// TIA Portal V18 export
FUNCTION "HC_PIDs" : Void   // FC1019, LAD
{ S7_Optimized_Access := 'TRUE' }
VERSION : 0.1
// stored: AutoNumber false, IsIECCheckEnabled false, SetENOAutomatically false, UDAEnableTagReadback false
BEGIN

REGION Network 1
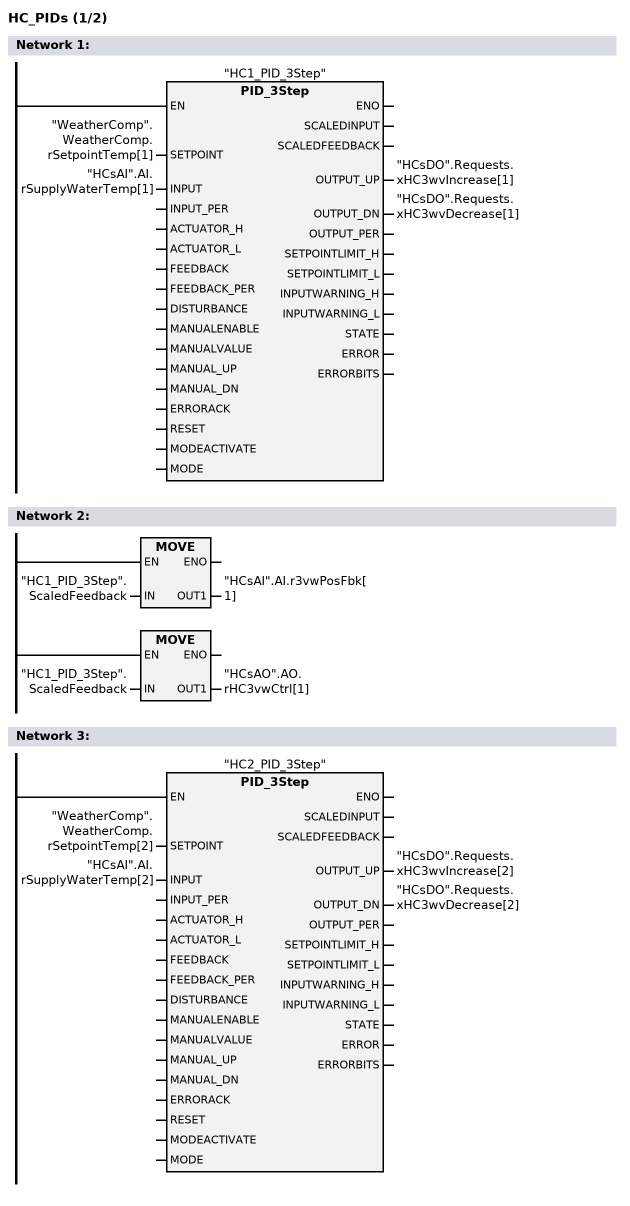
   RUNG wire#powerrail
      "HC1_PID_3Step".PID_3Step(Setpoint := "WeatherComp".WeatherComp.rSetpointTemp[1], Input := "HCsAI".AI.rSupplyWaterTemp[1], Input_PER :=, Actuator_H :=, Actuator_L :=, Feedback :=, Feedback_PER :=, Disturbance :=, ManualEnable :=, ManualValue :=, Manual_UP :=, Manual_DN :=, ErrorAck :=, Reset :=, ModeActivate :=, Mode :=, ScaledInput =>, ScaledFeedback =>, Output_UP => "HCsDO".Requests.xHC3wvIncrease[1], Output_DN => "HCsDO".Requests.xHC3wvDecrease[1], Output_PER =>, SetpointLimit_H =>, SetpointLimit_L =>, InputWarning_H =>, InputWarning_L =>, State =>, Error =>, ErrorBits =>)
   END_RUNG
   // the same network as SCL:
   "HC1_PID_3Step"(Setpoint := "WeatherComp".WeatherComp.rSetpointTemp[1],   // PID_3Step
                   Input := "HCsAI".AI.rSupplyWaterTemp[1],
                   Output_UP => "HCsDO".Requests.xHC3wvIncrease[1],
                   Output_DN => "HCsDO".Requests.xHC3wvDecrease[1]);
END_REGION

REGION Network 2
   RUNG wire#powerrail
      Move(in := "HC1_PID_3Step".ScaledFeedback, out1 => "HCsAI".AI.r3vwPosFbk[1])
   END_RUNG
   RUNG wire#powerrail
      Move(in := "HC1_PID_3Step".ScaledFeedback, out1 => "HCsAO".AO.rHC3vwCtrl[1])
   END_RUNG
   // the same network as SCL:
   "HCsAI".AI.r3vwPosFbk[1] := "HC1_PID_3Step".ScaledFeedback;
   "HCsAO".AO.rHC3vwCtrl[1] := "HC1_PID_3Step".ScaledFeedback;
END_REGION

REGION Network 3
   RUNG wire#powerrail
      "HC2_PID_3Step".PID_3Step(Setpoint := "WeatherComp".WeatherComp.rSetpointTemp[2], Input := "HCsAI".AI.rSupplyWaterTemp[2], Input_PER :=, Actuator_H :=, Actuator_L :=, Feedback :=, Feedback_PER :=, Disturbance :=, ManualEnable :=, ManualValue :=, Manual_UP :=, Manual_DN :=, ErrorAck :=, Reset :=, ModeActivate :=, Mode :=, ScaledInput =>, ScaledFeedback =>, Output_UP => "HCsDO".Requests.xHC3wvIncrease[2], Output_DN => "HCsDO".Requests.xHC3wvDecrease[2], Output_PER =>, SetpointLimit_H =>, SetpointLimit_L =>, InputWarning_H =>, InputWarning_L =>, State =>, Error =>, ErrorBits =>)
   END_RUNG
   // the same network as SCL:
   "HC2_PID_3Step"(Setpoint := "WeatherComp".WeatherComp.rSetpointTemp[2],   // PID_3Step
                   Input := "HCsAI".AI.rSupplyWaterTemp[2],
                   Output_UP => "HCsDO".Requests.xHC3wvIncrease[2],
                   Output_DN => "HCsDO".Requests.xHC3wvDecrease[2]);
END_REGION

REGION Network 4
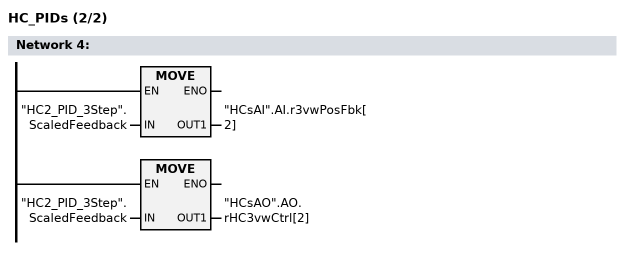
   RUNG wire#powerrail
      Move(in := "HC2_PID_3Step".ScaledFeedback, out1 => "HCsAI".AI.r3vwPosFbk[2])
   END_RUNG
   RUNG wire#powerrail
      Move(in := "HC2_PID_3Step".ScaledFeedback, out1 => "HCsAO".AO.rHC3vwCtrl[2])
   END_RUNG
   // the same network as SCL:
   "HCsAI".AI.r3vwPosFbk[2] := "HC2_PID_3Step".ScaledFeedback;
   "HCsAO".AO.rHC3vwCtrl[2] := "HC2_PID_3Step".ScaledFeedback;
END_REGION
END_FUNCTION
